# EPICS substitutions: iocs/bcur/iocBoot/iocbcur/substitutions/fb_epid.substitutions
# $Id$

file "$(OPTICS)/opticsApp/Db/fb_epid.db"
  {
    {
        P=bcur:epid1,
	IN=bcur:epid1:sim.VAL,
	OUT=bcur:epid1:sim.D,
	MODE=PID,
	CALC=A,
	PERMIT1="bcur:epid1:on.VAL",
	PERMIT2="",
	PERMIT3="",
	PERMIT4=""
    }
  }
